// SIMATIC STEP 7 (V5.x) project S_Pesaje
// CPU: CPU312(1)
// station: P_ADR_BUS
// station: Hardware
// station: Equipo SIMATIC 300
// program: Programa S7(1)

SYMBOL_TABLE
"PESAJE"	FC 2	FC 2	// Función de pesaje
"SCALE"	FC 105	FC 105	// Scaling Values
"BIT_DE_TRABAJO"	I 124.0	BOOL
"RECIBIDO"	I 124.1	BOOL
"START"	I 124.2	BOOL
"PESO_SARTEN"	MD 100	REAL
"PESO_CACEROLA"	MD 104	REAL
"PESO_WOK"	MD 108	REAL
"PESO_PAELLERA"	MD 112	REAL
"PESO"	MD 116	REAL
"Cycle Execution"	OB 1	OB 1
"IN"	PIW 651	INT
"STBY"	Q 100.0	BOOL
"SARTEN"	Q 100.1	BOOL
"CACEROLA"	Q 100.2	BOOL
"WOK"	Q 100.3	BOOL
"PAELLERA"	Q 100.4	BOOL
END_SYMBOL_TABLE

FUNCTION "PESAJE" : VOID	// FC 2
TITLE = PESAJE
VERSION : 0.1
VAR_INPUT
  in : INT ;
  PESO_SARTEN : REAL ;
  PESO_CACEROLA : REAL ;
  PESO_WOK : REAL ;
  PESO_PAELLERA : REAL ;
  bit_de_trabajo : BOOL ;
  RECIBIDO : BOOL ;
  START : BOOL ;
END_VAR
VAR_OUTPUT
  stby : BOOL ;
  SARTEN : BOOL ;
  CACEROLA : BOOL ;
  WOK : BOOL ;
  PAELLERA : BOOL ;
  PESO_OUT : REAL ;
END_VAR
VAR_TEMP
  retFC105 : WORD ;
  x121 : BOOL ;
  x122 : BOOL ;
  x123 : BOOL ;
  x124 : BOOL ;
  m3 : BOOL ;
  x120 : BOOL ;
  FP_BDT : BOOL ;
  FP_START : BOOL ;
  PESO : REAL ;
END_VAR
BEGIN
NETWORK
TITLE = Pesado
      A     #m3;
      CALL  "SCALE" (
           $1                       := #in,
           $2                       := L#1133903872,
           $3                       := L#0,
           $4                       := FALSE,
           $5                       := #retFC105,
           $6                       := #PESO);
NETWORK
TITLE =
      A     #x120;
      A     #START;
      FP    #FP_START;
      R     #x120;
      S     #m3;
NETWORK
TITLE = Arranque
      A     #bit_de_trabajo;
      FP    #FP_BDT;
      S     #x120;
      R     #m3;
      R     #x121;
      R     #x122;
      R     #x123;
      R     #x124;
NETWORK
TITLE =
      A(;
      L     #PESO_SARTEN;
      L     5.000000e+00;
      +R;
      L     #PESO;
      >R;
      );
      A(;
      L     #PESO_SARTEN;
      L     5.000000e+00;
      -R;
      L     #PESO;
      <R;
      );
      A     #m3;
      R     #m3;
      S     #x121;
NETWORK
TITLE =
      L     #PESO;
      T     #PESO_OUT;
NETWORK
TITLE =
      A(;
      L     #PESO_CACEROLA;
      L     5.000000e+00;
      +R;
      L     #PESO;
      >R;
      );
      A(;
      L     #PESO_CACEROLA;
      L     5.000000e+00;
      -R;
      L     #PESO;
      <R;
      );
      A     #m3;
      R     #m3;
      S     #x122;
NETWORK
TITLE =
      A(;
      L     #PESO_WOK;
      L     5.000000e+00;
      +R;
      L     #PESO;
      >R;
      );
      A(;
      L     #PESO_WOK;
      L     5.000000e+00;
      -R;
      L     #PESO;
      <R;
      );
      A     #m3;
      R     #m3;
      S     #x123;
NETWORK
TITLE =
      A(;
      L     #PESO_PAELLERA;
      L     5.000000e+00;
      +R;
      L     #PESO;
      >R;
      );
      A(;
      L     #PESO_PAELLERA;
      L     5.000000e+00;
      -R;
      L     #PESO;
      <R;
      );
      A     #m3;
      R     #m3;
      S     #x124;
NETWORK
TITLE = TRATAMIENTO SALIDAS
      A     #x121;
      =     #SARTEN;
      A     #x122;
      =     #CACEROLA;
      A     #x123;
      =     #WOK;
      A     #x124;
      =     #PAELLERA;
      A     #x120;
      =     #stby;
NETWORK
TITLE = Paso de estado pesado a stby
      A(;
      A     #x121;
      O     #x122;
      O     #x123;
      O     #x124;
      );
      A     #RECIBIDO;
      R     #x121;
      R     #x122;
      R     #x123;
      R     #x124;
      S     #x120;
END_FUNCTION

// FC 105: know-how protected block, not included

ORGANIZATION_BLOCK "Cycle Execution"	// OB 1
TITLE = "Main Program Sweep (Cycle)"
VERSION : 0.1
VAR_TEMP
  OB1_EV_CLASS : BYTE ;	//Bits 0-3 = 1 (Coming event), Bits 4-7 = 1 (Event class 1)
  OB1_SCAN_1 : BYTE ;	//1 (Cold restart scan 1 of OB 1), 3 (Scan 2-n of OB 1)
  OB1_PRIORITY : BYTE ;	//Priority of OB Execution
  OB1_OB_NUMBR : BYTE ;	//1 (Organization block 1, OB1)
  OB1_RESERVED_1 : BYTE ;	//Reserved for system
  OB1_RESERVED_2 : BYTE ;	//Reserved for system
  OB1_PREV_CYCLE : INT ;	//Cycle time of previous OB1 scan (milliseconds)
  OB1_MIN_CYCLE : INT ;	//Minimum cycle time of OB1 (milliseconds)
  OB1_MAX_CYCLE : INT ;	//Maximum cycle time of OB1 (milliseconds)
  OB1_DATE_TIME : DATE_AND_TIME ;	//Date and time OB1 started
END_VAR
BEGIN
NETWORK
TITLE =
      CALL  "PESAJE" (
           in                       := "IN",
           PESO_SARTEN              := "PESO_SARTEN",
           PESO_CACEROLA            := "PESO_CACEROLA",
           PESO_WOK                 := "PESO_WOK",
           PESO_PAELLERA            := "PESO_PAELLERA",
           bit_de_trabajo           := "BIT_DE_TRABAJO",
           RECIBIDO                 := "RECIBIDO",
           START                    := "START",
           stby                     := "STBY",
           SARTEN                   := "SARTEN",
           CACEROLA                 := "CACEROLA",
           WOK                      := "WOK",
           PAELLERA                 := "PAELLERA",
           PESO_OUT                 := "PESO");
END_ORGANIZATION_BLOCK
